FUNCTION_BLOCK Watertank
  (* Standard: 61499-2 *)
  (* Version 0,1, 2015-00-07, Th?o, PC_THEO *)
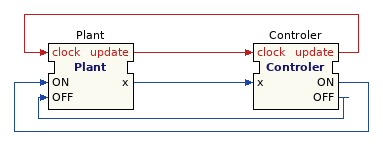
  FBS
    Plant : Plant;
    Controler : Controler;
  END_FBS
  EVENT_CONNECTIONS
    Plant.update TO Controler.clock;
    Controler.update TO Plant.clock;
  END_CONNECTIONS
  DATA_CONNECTIONS
    Plant.x TO Controler.x;
    Controler.ON TO Plant.ON;
    Controler.OFF TO Plant.OFF;
  END_CONNECTIONS
END_FUNCTION_BLOCK
